# EPICS StreamDevice protocol: stanfordDG645/stanfordDG645.proto
# Protocol file for Stanford Digital Delay Generator DG645

ReplyTimeout = 1000;
Terminator = CR LF;

getDelay {
         out "DLAY?\$1";
         in "%*u,%f";
}

setDelay {
         out "DLAY \$1,\$2,%e";
         out "*WAI";
         out "LERR?";
         in "0";
}
